PROGRAM MAIN
VAR
	// Simple establishing of core variables
	bStartbutton : BOOL := FALSE;
	bStopbutton : BOOL := FALSE;

	bConveyoron : BOOL := FALSE;
END_VAR

// This is a simple code that starts and stops a virtual belt depending on which button is being pressed while resetting the button inputs after each signal.
bConveyoron := (bStartbutton OR bConveyoron) AND NOT bStopbutton;
IF bStartbutton := TRUE THEN
	bStopbutton := FALSE;
	bStartbutton := FALSE;
END_IF;
IF bStopbutton := TRUE THEN
	bStopbutton := FALSE;
	bStartbutton := FALSE;
END_IF;

END_PROGRAM

(* stored: Version 1.1.0.1, ProductVersion 3.1.4024.16
   POU MAIN: Id {116e7d30-b956-4213-8d9a-f39d94a2d40c}, SpecialFunc None *)
